Universal Robots PolyScope program: gripper_23.urp

Program gripper_23 (installation=default directory=/programs/usbdisk/nova pasta createdIn=5.10.0.106288 lastSavedIn=5.10.0.106288 robotSerialNumber=20205501854)
Calibrated DH parameters: a=[0.000184, -0.272509, -0.38425, 0.000028, 0.000032, 0]; d=[0.162742, -337.661697, 348.3844, -10.588954, 0.099709, 0.09958]; alpha=[1.571678, -0.000966, 0.007363, 1.569932, -1.570277, 0]; deltaTheta=[0, 0.875055, 5.610779, -0.202656, -0.000001, 0]
Robot Program (runOnlyOnce=false)
  URCap SCHUNK EGH Gripper (SCHUNK Gripper, SCHUNK GmbH & Co. KG) dataModel(Defined=false, command=4, pdGripDirection=1, forceSave=15, waitforcompletion=true)
  URCap SCHUNK EGH Gripper (SCHUNK Gripper, SCHUNK GmbH & Co. KG) dataModel(Defined=false, pdGripTargetPosition=20.3, command=7, waitforcompletion=true, pdTargetPosition=23.0, pdGripDirection=1, forceSave=140)
